# EPICS StreamDevice protocol: apps/chillerApp/Db/Lauda_XT.proto
#
# Lauda Integral XT Series process thermostats
#
# Parameters:
#   $1 = input channel number [1-8]
#
# Author: Wesley Moore
# Date:   December 2015
#

OutTerminator = CR LF;
InTerminator = CR LF;
writetimeout = 100;
readtimeout = 300;     # milliseconds
replytimeout = 1000;
ExtraInput = Ignore;

###################################
# INPUTS
###################################
getAi {
	out "\$1";
    in "%f";
}

getBi {
    out "\$1";
    in "%d";
}

getMbbi {
    out "\$1";
    in "%b";
}

###################################
# OUTPUTS
###################################
setAo {
	out "\$1_%.3f";
    in "OK";
}

setAoInit {
	out "OUT_\$1_%.3f";
    in "OK";
    @init {
        out "IN_\$1";
        in "%f";
    }
}

setMbbo {
    out "\$1_%d";
    in "OK";
}

writeStr {
    out "\$1";
}
